{attribute addProperty BoxType "EL1502--0000"}
{attribute addProperty Id "CNT_InputsAT %I*CNT_Inputs_2DD1A21088110CNT_OutputsAT %Q*CNT_Outputs_5A50AE9A6480WcStateAT %I*WcState_98A4DF7520.250InfoDataAT %I*InfoData_BC63D37F80100"}
{attribute addProperty CRC "2242762266"}
{attribute addProperty SizeInBites "234"}
{attribute addProperty SizeInBytes "29.25"}
TYPE EL1502_BA17F412 :
STRUCT
	{attribute addProperty Name "CNT_Inputs"}
	CNT_Inputs : CNT_Inputs_2DD1A210;
	{attribute addProperty Name "CNT_Outputs"}
	CNT_Outputs : CNT_Outputs_5A50AE9A;
	{attribute addProperty Name "WcState"}
	WcState : WcState_98A4DF75;
	{attribute addProperty Name "InfoData"}
	InfoData : InfoData_BC63D37F;
END_STRUCT
END_TYPE

(* stored: Version 1.2.0.0, ProductVersion 3.1.4024.9
   DUT EL1502_BA17F412: Id {e9d14b23-73de-4d03-a249-39fa714a2714} *)
